Fanuc KAREL source: kb00165.KL

-- PROVISIONAL review KL for V770-1; original PC SHA256 44b02ff93d4f59f1e52da24a13c24f87915cad5d1bed431c10fdd9ddf0feaeb7
-- Incomplete behavior may be omitted. Consult companion uncertainty JSON. Do not deploy.
PROGRAM KB00165
%NOLOCKGROUP
BEGIN
  -- UNRESOLVED_PC offsets 5-12; opcodes 9D,23
  -- UNRESOLVED_PC offsets 17-24; opcodes 9D,23
  -- UNRESOLVED_PC offsets 29-36; opcodes 9D,23
  -- UNRESOLVED_PC offsets 41-63; opcodes 27,22,22,22,31
  -- UNRESOLVED_PC offsets 68-72; opcodes 7F
END KB00165
